// TIA Portal V18 export
FUNCTION_BLOCK "SideShifter_Hydraulic"   // FB4, LAD
{ S7_Optimized_Access := 'TRUE' }
// stored: MemoryReserve 100, SetENOAutomatically false
   VAR_INPUT
      Actuators_Down : Bool;
      Actuators_Up : Bool;
      Hydraulic_Unit : Bool;
      iAct1_1_Sensor_Up : Bool;
      iAct1_1_Sensor_Down : Bool;
      iAct1_2_Sensor_Up : Bool;
      iAct1_2_Sensor_Down : Bool;
   END_VAR
   VAR_OUTPUT
      oValve1_Up : Bool;
      oValve1_Down : Bool;
      oHydraulic_Unit : Bool;
   END_VAR
BEGIN

REGION Network 1
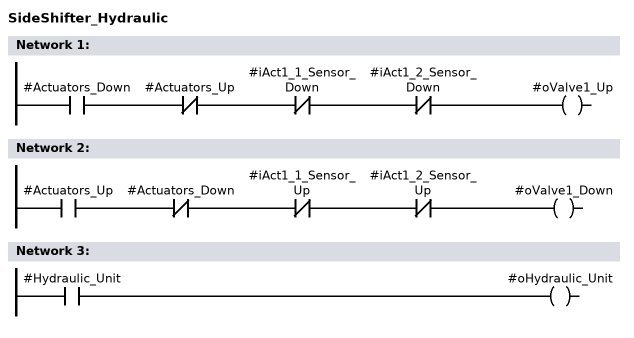
   RUNG wire#powerrail
      Contact( #Actuators_Down )
      I_Contact( #Actuators_Up )
      I_Contact( #iAct1_1_Sensor_Down )
      I_Contact( #iAct1_2_Sensor_Down )
      Coil( #oValve1_Up )
   END_RUNG
   // the same network as SCL:
   #oValve1_Up := #Actuators_Down AND NOT #Actuators_Up AND NOT #iAct1_1_Sensor_Down AND NOT #iAct1_2_Sensor_Down;
END_REGION

REGION Network 2
   RUNG wire#powerrail
      Contact( #Actuators_Up )
      I_Contact( #Actuators_Down )
      I_Contact( #iAct1_1_Sensor_Up )
      I_Contact( #iAct1_2_Sensor_Up )
      Coil( #oValve1_Down )
   END_RUNG
   // the same network as SCL:
   #oValve1_Down := #Actuators_Up AND NOT #Actuators_Down AND NOT #iAct1_1_Sensor_Up AND NOT #iAct1_2_Sensor_Up;
END_REGION

REGION Network 3
   RUNG wire#powerrail
      Contact( #Hydraulic_Unit )
      Coil( #oHydraulic_Unit )
   END_RUNG
   // the same network as SCL:
   #oHydraulic_Unit := #Hydraulic_Unit;
END_REGION
END_FUNCTION_BLOCK
